TYPE ST_AxisPersistent :
STRUCT

    iPositionAtShutdown : LREAL;
    bMovingAtShutdown   : BOOL;

END_STRUCT
END_TYPE

(* stored: Version 1.1.0.1, ProductVersion 3.1.4024.0
   DUT ST_AxisPersistent: Id {98d769cd-5416-4343-814a-f5a739d71156} *)
